{attribute 'qualified_only'}
{attribute 'to_string'}
TYPE ZAppStep :
(
  Undefined := 0
  
  ,BootBegin
  ,BootLoadDefaultData
  ,BootEnd
  ,BootFaultBegin
  ,BootFaultEnd 
  ,RunningBegin
  ,RunningEnd   
);
END_TYPE

(* stored: Version 1.1.0.1
   DUT ZAppStep: Id {8e834998-7ae4-423d-a589-1fbb41ef4d69} *)
